// TIA Portal V19 export
TYPE "LubrMotor_Alr"
// stored: Access Published
   STRUCT
      RotationFeedback : Bool;
      LowLevelLubrication : Bool;
      MotorAlr : "MotorAlr";
   END_STRUCT;
END_TYPE
